PROGRAM MAIN
VAR
END_VAR

END_PROGRAM

(* stored: Version 1.1.0.1
   POU MAIN: Id {0a93f00b-5218-452b-bb0b-68f177a76102} *)
